// TIA Portal project "LinkedList_v000_000_002" (V16)
// task for 000.000.002: create LinkedList.FindAvailableSlot()

(* hardware
DEVICE "S7-1200 station_1"  S7-1200 Station
   slot 0: "Rack_0"  S7-1200 Rack  Rack  V1.0
   slot 1: "PLC_1"  CPU 1212C DC/DC/DC  6ES7 212-1AE40-0XB0  V4.4
*)

// ===== PLC "PLC_1"  CPU 1212C DC/DC/DC =====

VAR_GLOBAL   // PLC tag table "Default tag table"
   "System_Byte" AT %MB1 : Byte;
   "FirstScan" AT %M1.0 : Bool;
   "DiagStatusUpdate" AT %M1.1 : Bool;
   "AlwaysTRUE" AT %M1.2 : Bool;
   "AlwaysFALSE" AT %M1.3 : Bool;
   "Clock_Byte" AT %MB0 : Byte;
   "Clock_10Hz" AT %M0.0 : Bool;
   "Clock_5Hz" AT %M0.1 : Bool;
   "Clock_2.5Hz" AT %M0.2 : Bool;
   "Clock_2Hz" AT %M0.3 : Bool;
   "Clock_1.25Hz" AT %M0.4 : Bool;
   "Clock_1Hz" AT %M0.5 : Bool;
   "Clock_0.625Hz" AT %M0.6 : Bool;
   "Clock_0.5Hz" AT %M0.7 : Bool;
END_VAR

TYPE "LinkedList.Node.Payload.UDT"
   STRUCT
      id : Char;
      status : String;
   END_STRUCT;
END_TYPE

TYPE "LinkedList.Node.UDT"
   STRUCT
      payload : "LinkedList.Node.Payload.UDT";
      pointer : DInt;
   END_STRUCT;
END_TYPE

TYPE "LinkedList.UDT"
   STRUCT
      head : DInt;
      list : Array[0..4] of "LinkedList.Node.UDT";
   END_STRUCT;
END_TYPE

FUNCTION_BLOCK "LinkedList"   // FB1, SCL
TITLE = Linked List
{ S7_Optimized_Access := 'TRUE' }
AUTHOR : Machado
FAMILY : LinkedList
VERSION : 0.1
   VAR
      list : "LinkedList.UDT";
   END_VAR
BEGIN
END_FUNCTION_BLOCK

FUNCTION "LinkedList.FindPointer" : DInt   // FC1, SCL
TITLE = Find Node in a Linked List by Pointer
{ S7_Optimized_Access := 'TRUE' }
AUTHOR : Machado
FAMILY : LinkedList
VERSION : 0.1
   VAR_INPUT
      needle : "LinkedList.Node.Payload.UDT";
      not_found : DInt;
   END_VAR
   VAR_IN_OUT
      list : Array[*] of "LinkedList.Node.UDT";
   END_VAR
   VAR_TEMP
      i : DInt;
      size : DInt;
   END_VAR
BEGIN
   #size := UDINT_TO_DINT("LinkedList.Node[].CountOfElements"(#list));

   FOR #i := 0 TO #size - 1 DO
       IF #list[#i].payload <> #needle THEN
           CONTINUE;
       END_IF;
       #"LinkedList.FindPointer" := #i;
       RETURN;
   END_FOR;

   #"LinkedList.FindPointer" := #not_found;
   RETURN;
END_FUNCTION

FUNCTION "LinkedList.FindPayload" : DInt   // FC1, SCL
TITLE = Find Node in a Linked List by Payload
{ S7_Optimized_Access := 'TRUE' }
AUTHOR : Machado
FAMILY : LinkedList
VERSION : 0.1
   VAR_INPUT
      needle : DInt;
      not_found : DInt;
   END_VAR
   VAR_IN_OUT
      list : Array[*] of "LinkedList.Node.UDT";
   END_VAR
   VAR_TEMP
      i : DInt;
      size : DInt;
   END_VAR
BEGIN
   #size := UDINT_TO_DINT("LinkedList.Node[].CountOfElements"(#list));

   FOR #i := 0 TO #size - 1 DO
       IF #list[#i]."pointer" <> #needle THEN
           CONTINUE;
       END_IF;
       #"LinkedList.FindPointer" := #i;
       RETURN;
   END_FOR;

   #"LinkedList.FindPointer" := #not_found;
   RETURN;
END_FUNCTION

FUNCTION "LinkedList.FindID" : DInt   // FC1, SCL
TITLE = Find Node in a Linked List by Payload
{ S7_Optimized_Access := 'TRUE' }
AUTHOR : Machado
FAMILY : LinkedList
VERSION : 0.1
   VAR_INPUT
      needle : Char;
      not_found : DInt;
   END_VAR
   VAR_IN_OUT
      list : Array[*] of "LinkedList.Node.UDT";
   END_VAR
   VAR_TEMP
      i : DInt;
      size : DInt;
   END_VAR
BEGIN
   #size := UDINT_TO_DINT("LinkedList.Node[].CountOfElements"(#list));

   FOR #i := 0 TO #size - 1 DO
       IF #list[#i].payload.id <> #needle THEN
           CONTINUE;
       END_IF;
       #"LinkedList.FindID" := #i;
       RETURN;
   END_FOR;

   #"LinkedList.FindID" := #not_found;
   RETURN;
END_FUNCTION

FUNCTION "LinkedList.FindStatus" : DInt   // FC1, SCL
TITLE = Find Node in a Linked List by Payload
{ S7_Optimized_Access := 'TRUE' }
AUTHOR : Machado
FAMILY : LinkedList
VERSION : 0.1
   VAR_INPUT
      needle : String;
      not_found : DInt;
   END_VAR
   VAR_IN_OUT
      list : Array[*] of "LinkedList.Node.UDT";
   END_VAR
   VAR_TEMP
      i : DInt;
      size : DInt;
   END_VAR
BEGIN
   #size := UDINT_TO_DINT("LinkedList.Node[].CountOfElements"(#list));

   FOR #i := 0 TO #size - 1 DO
       IF #list[#i].payload.status <> #needle THEN
           CONTINUE;
       END_IF;
       #"LinkedList.FindStatus" := #i;
       RETURN;
   END_FOR;

   #"LinkedList.FindStatus" := #not_found;
   RETURN;
END_FUNCTION

FUNCTION "LinkedList.Node[].CountOfElements" : UDInt   // FC2, SCL
TITLE = Count of Elements of an Array of Link List Nodes
{ S7_Optimized_Access := 'TRUE' }
AUTHOR : Machado
FAMILY : LinkedList
VERSION : 0.1
   VAR_INPUT
      list : Variant;
   END_VAR
BEGIN
   #"LinkedList.Node[].CountOfElements" := CountOfElements(#list);
   RETURN;
END_FUNCTION

ORGANIZATION_BLOCK "Main"   // OB1, LAD, ProgramCycle
TITLE = "Main Program Sweep (Cycle)"
{ S7_Optimized_Access := 'TRUE' }
VERSION : 0.1
   VAR_INPUT
      Initial_Call : Bool;   // Initial call of this OB
      Remanence : Bool;   // =True, if remanent data are available
   END_VAR
BEGIN
END_ORGANIZATION_BLOCK